PROGRAM MAIN
VAR
    fbTimer: TON;
END_VAR

(*
Millis (1 regel code)

Maak met slechts één FB een programma dat iedere x milliseconden één enkele puls geeft.
*)

fbTimer(IN:=NOT fbTimer.Q, PT:=T#3ms);

END_PROGRAM

(* stored: Version 1.1.0.1, ProductVersion 3.1.4024.12
   POU MAIN: Id {3858e7b4-116a-41cb-9324-bee8c68304bb}, SpecialFunc None *)
